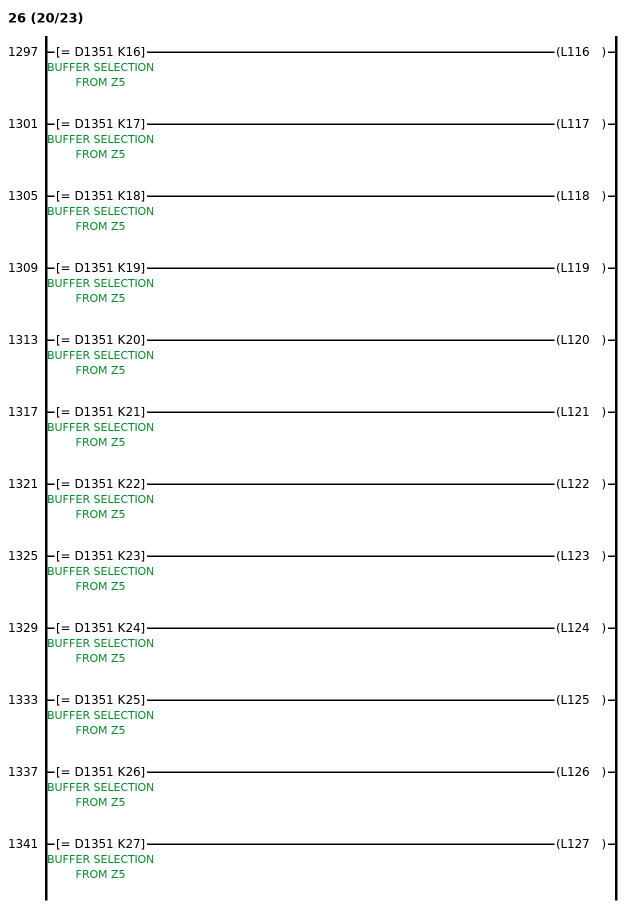
1297  LD=     D1351 K16  ; BUFFER SELECTION FROM Z5
      OUT     L116
1301  LD=     D1351 K17  ; BUFFER SELECTION FROM Z5
      OUT     L117
1305  LD=     D1351 K18  ; BUFFER SELECTION FROM Z5
      OUT     L118
1309  LD=     D1351 K19  ; BUFFER SELECTION FROM Z5
      OUT     L119
1313  LD=     D1351 K20  ; BUFFER SELECTION FROM Z5
      OUT     L120
1317  LD=     D1351 K21  ; BUFFER SELECTION FROM Z5
      OUT     L121
1321  LD=     D1351 K22  ; BUFFER SELECTION FROM Z5
      OUT     L122
1325  LD=     D1351 K23  ; BUFFER SELECTION FROM Z5
      OUT     L123
1329  LD=     D1351 K24  ; BUFFER SELECTION FROM Z5
      OUT     L124
1333  LD=     D1351 K25  ; BUFFER SELECTION FROM Z5
      OUT     L125
1337  LD=     D1351 K26  ; BUFFER SELECTION FROM Z5
      OUT     L126
1341  LD=     D1351 K27  ; BUFFER SELECTION FROM Z5
      OUT     L127
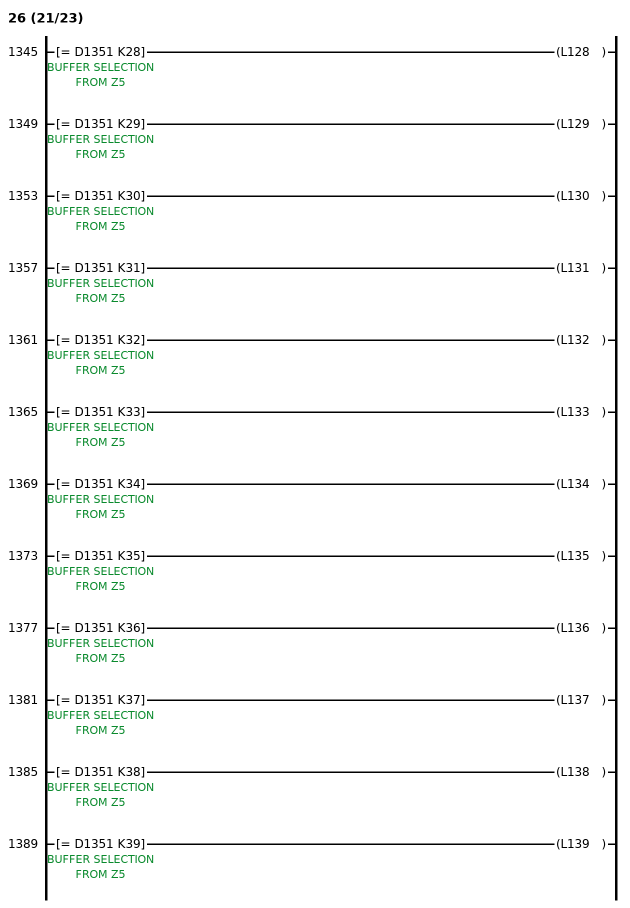
1345  LD=     D1351 K28  ; BUFFER SELECTION FROM Z5
      OUT     L128
1349  LD=     D1351 K29  ; BUFFER SELECTION FROM Z5
      OUT     L129
1353  LD=     D1351 K30  ; BUFFER SELECTION FROM Z5
      OUT     L130
1357  LD=     D1351 K31  ; BUFFER SELECTION FROM Z5
      OUT     L131
1361  LD=     D1351 K32  ; BUFFER SELECTION FROM Z5
      OUT     L132
1365  LD=     D1351 K33  ; BUFFER SELECTION FROM Z5
      OUT     L133
1369  LD=     D1351 K34  ; BUFFER SELECTION FROM Z5
      OUT     L134
1373  LD=     D1351 K35  ; BUFFER SELECTION FROM Z5
      OUT     L135
1377  LD=     D1351 K36  ; BUFFER SELECTION FROM Z5
      OUT     L136
1381  LD=     D1351 K37  ; BUFFER SELECTION FROM Z5
      OUT     L137
1385  LD=     D1351 K38  ; BUFFER SELECTION FROM Z5
      OUT     L138
1389  LD=     D1351 K39  ; BUFFER SELECTION FROM Z5
      OUT     L139
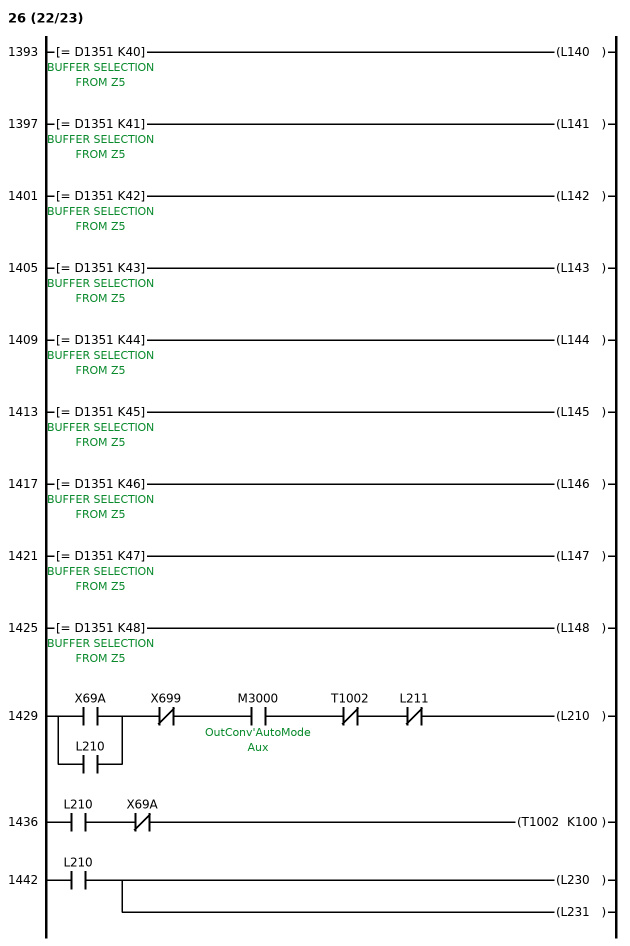
1393  LD=     D1351 K40  ; BUFFER SELECTION FROM Z5
      OUT     L140
1397  LD=     D1351 K41  ; BUFFER SELECTION FROM Z5
      OUT     L141
1401  LD=     D1351 K42  ; BUFFER SELECTION FROM Z5
      OUT     L142
1405  LD=     D1351 K43  ; BUFFER SELECTION FROM Z5
      OUT     L143
1409  LD=     D1351 K44  ; BUFFER SELECTION FROM Z5
      OUT     L144
1413  LD=     D1351 K45  ; BUFFER SELECTION FROM Z5
      OUT     L145
1417  LD=     D1351 K46  ; BUFFER SELECTION FROM Z5
      OUT     L146
1421  LD=     D1351 K47  ; BUFFER SELECTION FROM Z5
      OUT     L147
1425  LD=     D1351 K48  ; BUFFER SELECTION FROM Z5
      OUT     L148
1429  LD      X69A
      OR      L210
      ANI     X699
      AND     M3000  ; OutConv'AutoModeAux
      ANI     T1002
      ANI     L211
      OUT     L210
1436  LD      L210
      ANI     X69A
      OUT     T1002 K100
1442  LD      L210
      OUT     L230
      OUT     L231
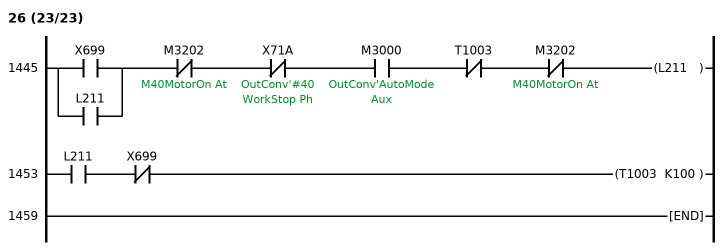
1445  LD      X699
      OR      L211
      ANI     M3202  ; M40MotorOn At
      ANI     X71A  ; OutConv'#40 WorkStop Ph
      AND     M3000  ; OutConv'AutoModeAux
      ANI     T1003
      ANI     M3202  ; M40MotorOn At
      OUT     L211
1453  LD      L211
      ANI     X699
      OUT     T1003 K100
1459  END
END_PROGRAM

PROGRAM 30  // Cycle Time
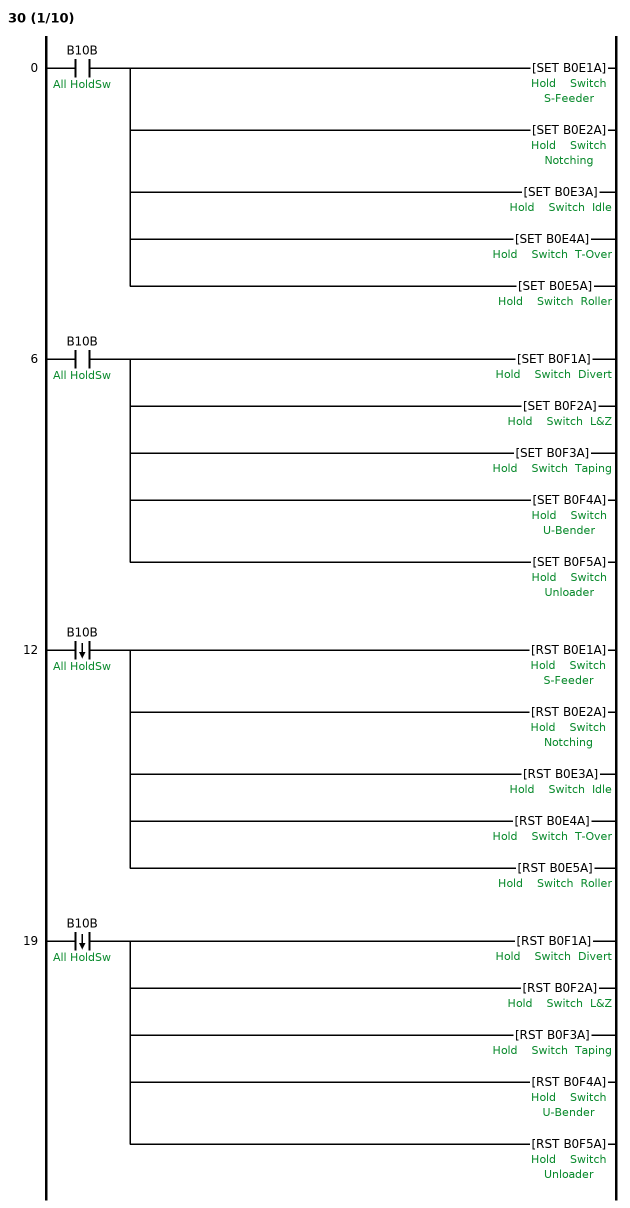
0     LD      B10B  ; All HoldSw
      SET     B0E1A  ; Hold    Switch  S-Feeder
      SET     B0E2A  ; Hold    Switch  Notching
      SET     B0E3A  ; Hold    Switch  Idle
      SET     B0E4A  ; Hold    Switch  T-Over
      SET     B0E5A  ; Hold    Switch  Roller
6     LD      B10B  ; All HoldSw
      SET     B0F1A  ; Hold    Switch  Divert
      SET     B0F2A  ; Hold    Switch  L&Z
      SET     B0F3A  ; Hold    Switch  Taping
      SET     B0F4A  ; Hold    Switch  U-Bender
      SET     B0F5A  ; Hold    Switch  Unloader
12    LDF     B10B  ; All HoldSw
      RST     B0E1A  ; Hold    Switch  S-Feeder
      RST     B0E2A  ; Hold    Switch  Notching
      RST     B0E3A  ; Hold    Switch  Idle
      RST     B0E4A  ; Hold    Switch  T-Over
      RST     B0E5A  ; Hold    Switch  Roller
19    LDF     B10B  ; All HoldSw
      RST     B0F1A  ; Hold    Switch  Divert
      RST     B0F2A  ; Hold    Switch  L&Z
      RST     B0F3A  ; Hold    Switch  Taping
      RST     B0F4A  ; Hold    Switch  U-Bender
      RST     B0F5A  ; Hold    Switch  Unloader
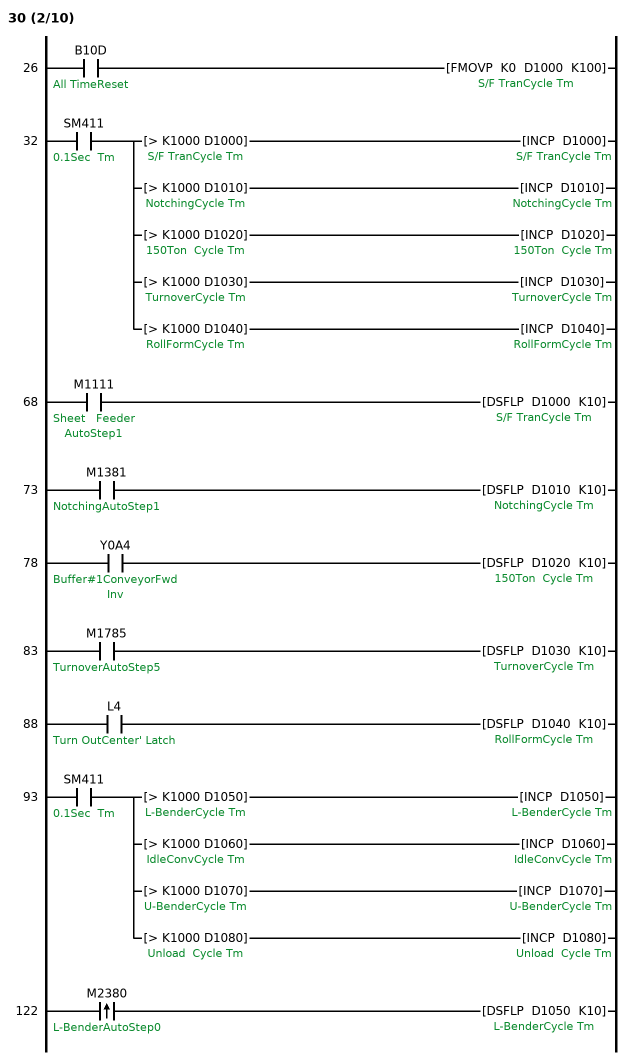
26    LD      B10D  ; All TimeReset
      FMOVP   K0 D1000 K100  ; S/F TranCycle Tm
32    LD      SM411  ; 0.1Sec  Tm
      MPS
      AND>    K1000 D1000  ; S/F TranCycle Tm
      INCP    D1000
      MRD
      AND>    K1000 D1010  ; NotchingCycle Tm
      INCP    D1010
      MRD
      AND>    K1000 D1020  ; 150Ton  Cycle Tm
      INCP    D1020
      MRD
      AND>    K1000 D1030  ; TurnoverCycle Tm
      INCP    D1030
      MPP
      AND>    K1000 D1040  ; RollFormCycle Tm
      INCP    D1040
68    LD      M1111  ; Sheet   Feeder  AutoStep1
      DSFLP   D1000 K10
73    LD      M1381  ; NotchingAutoStep1
      DSFLP   D1010 K10
78    LD      Y0A4  ; Buffer#1ConveyorFwd Inv
      DSFLP   D1020 K10
83    LD      M1785  ; TurnoverAutoStep5
      DSFLP   D1030 K10
88    LD      L4  ; Turn OutCenter' Latch
      DSFLP   D1040 K10
93    LD      SM411  ; 0.1Sec  Tm
      MPS
      AND>    K1000 D1050  ; L-BenderCycle Tm
      INCP    D1050
      MRD
      AND>    K1000 D1060  ; IdleConvCycle Tm
      INCP    D1060
      MRD
      AND>    K1000 D1070  ; U-BenderCycle Tm
      INCP    D1070
      MPP
      AND>    K1000 D1080  ; Unload  Cycle Tm
      INCP    D1080
122   LDP     M2380  ; L-BenderAutoStep0
      DSFLP   D1050 K10
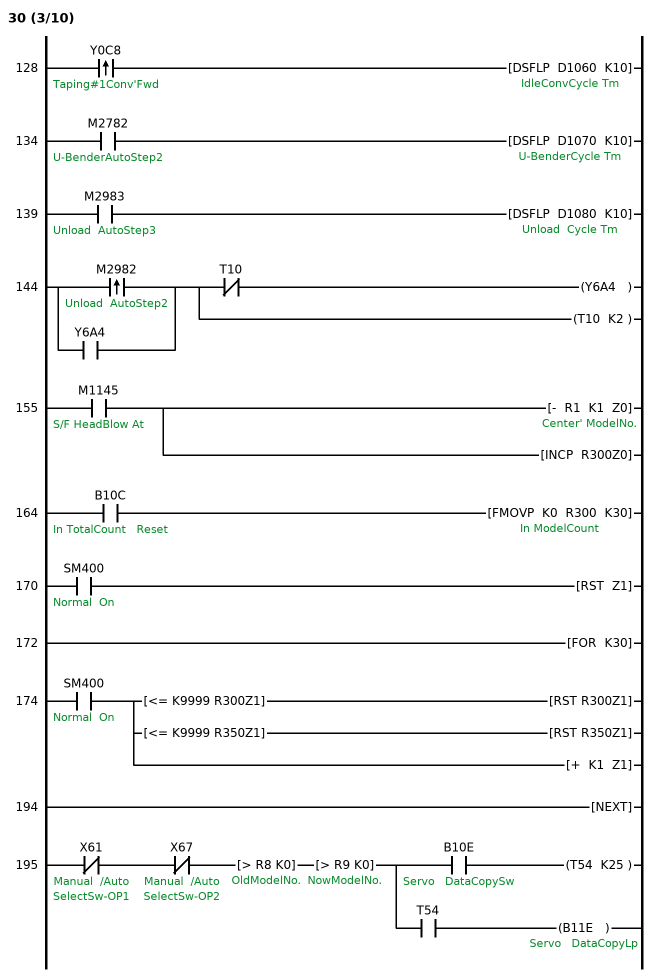
128   LDP     Y0C8  ; Taping#1Conv'Fwd
      DSFLP   D1060 K10
134   LD      M2782  ; U-BenderAutoStep2
      DSFLP   D1070 K10
139   LD      M2983  ; Unload  AutoStep3
      DSFLP   D1080 K10
144   LDP     M2982  ; Unload  AutoStep2
      OR      Y6A4
      MPS
      ANI     T10
      OUT     Y6A4
      MPP
      OUT     T10 K2
155   LD      M1145  ; S/F HeadBlow At
      -       R1 K1 Z0  ; Center' ModelNo.
      INCP    R300Z0
164   LD      B10C  ; In TotalCount   Reset
      FMOVP   K0 R300 K30  ; In ModelCount
170   LD      SM400  ; Normal  On
      RST     Z1
172   FOR     K30
174   LD      SM400  ; Normal  On
      MPS
      AND<=   K9999 R300Z1
      RST     R300Z1
      MRD
      AND<=   K9999 R350Z1
      RST     R350Z1
      MPP
      +       K1 Z1
194   NEXT
195   LDI     X61  ; Manual  /Auto   SelectSw-OP1
      ANI     X67  ; Manual  /Auto   SelectSw-OP2
      AND>    R8 K0  ; OldModelNo.
      AND>    R9 K0  ; NowModelNo.
      MPS
      AND     B10E  ; Servo   DataCopySw
      OUT     T54 K25
      MPP
      AND     T54
      OUT     B11E  ; Servo   DataCopyLp
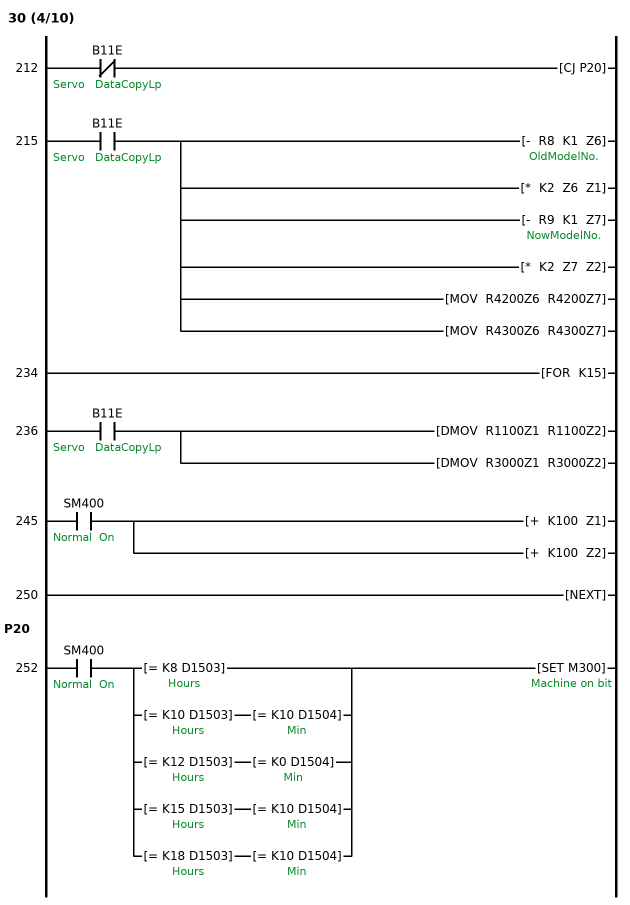
212   LDI     B11E  ; Servo   DataCopyLp
      CJ      P20
215   LD      B11E  ; Servo   DataCopyLp
      -       R8 K1 Z6
      *       K2 Z6 Z1
      -       R9 K1 Z7
      *       K2 Z7 Z2
      MOV     R4200Z6 R4200Z7
      MOV     R4300Z6 R4300Z7
234   FOR     K15
236   LD      B11E  ; Servo   DataCopyLp
      DMOV    R1100Z1 R1100Z2
      DMOV    R3000Z1 R3000Z2
245   LD      SM400  ; Normal  On
      +       K100 Z1
      +       K100 Z2
250   NEXT
      P20
252   LD      SM400  ; Normal  On
      LD=     K8 D1503  ; Hours
      LD=     K10 D1503  ; Hours
      AND=    K10 D1504  ; Min
      ORB
      LD=     K12 D1503  ; Hours
      AND=    K0 D1504  ; Min
      ORB
      LD=     K15 D1503  ; Hours
      AND=    K10 D1504  ; Min
      ORB
      LD=     K18 D1503  ; Hours
      AND=    K10 D1504  ; Min
      ORB
      ANB
      SET     M300  ; Machine on bit
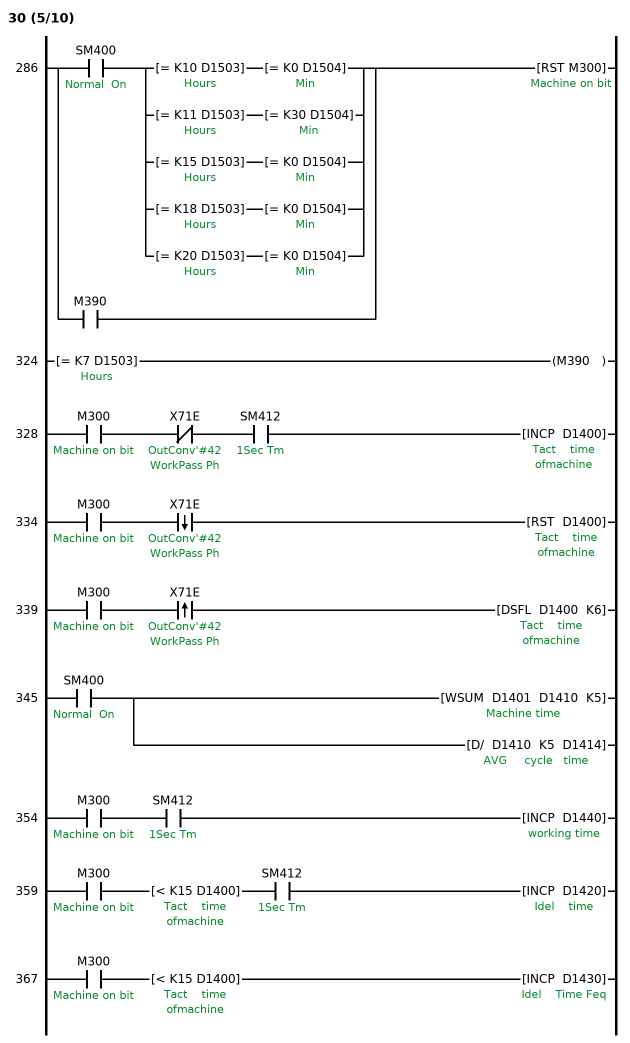
286   LD      SM400  ; Normal  On
      LD=     K10 D1503  ; Hours
      AND=    K0 D1504  ; Min
      LD=     K11 D1503  ; Hours
      AND=    K30 D1504  ; Min
      ORB
      LD=     K15 D1503  ; Hours
      AND=    K0 D1504  ; Min
      ORB
      LD=     K18 D1503  ; Hours
      AND=    K0 D1504  ; Min
      ORB
      LD=     K20 D1503  ; Hours
      AND=    K0 D1504  ; Min
      ORB
      ANB
      OR      M390
      RST     M300  ; Machine on bit
324   LD=     K7 D1503  ; Hours
      OUT     M390
328   LD      M300  ; Machine on bit
      ANI     X71E  ; OutConv'#42 WorkPass Ph
      AND     SM412  ; 1Sec Tm
      INCP    D1400  ; Tact    time  ofmachine
334   LD      M300  ; Machine on bit
      ANDF    X71E  ; OutConv'#42 WorkPass Ph
      RST     D1400  ; Tact    time  ofmachine
339   LD      M300  ; Machine on bit
      ANDP    X71E  ; OutConv'#42 WorkPass Ph
      DSFL    D1400 K6
345   LD      SM400  ; Normal  On
      WSUM    D1401 D1410 K5  ; Machine time
      D/      D1410 K5 D1414  ; AVG     cycle   time
354   LD      M300  ; Machine on bit
      AND     SM412  ; 1Sec Tm
      INCP    D1440  ; working time
359   LD      M300  ; Machine on bit
      AND<    K15 D1400  ; Tact    time  ofmachine
      AND     SM412  ; 1Sec Tm
      INCP    D1420  ; Idel    time
367   LD      M300  ; Machine on bit
      AND<    K15 D1400  ; Tact    time  ofmachine
      INCP    D1430  ; Idel    Time Feq
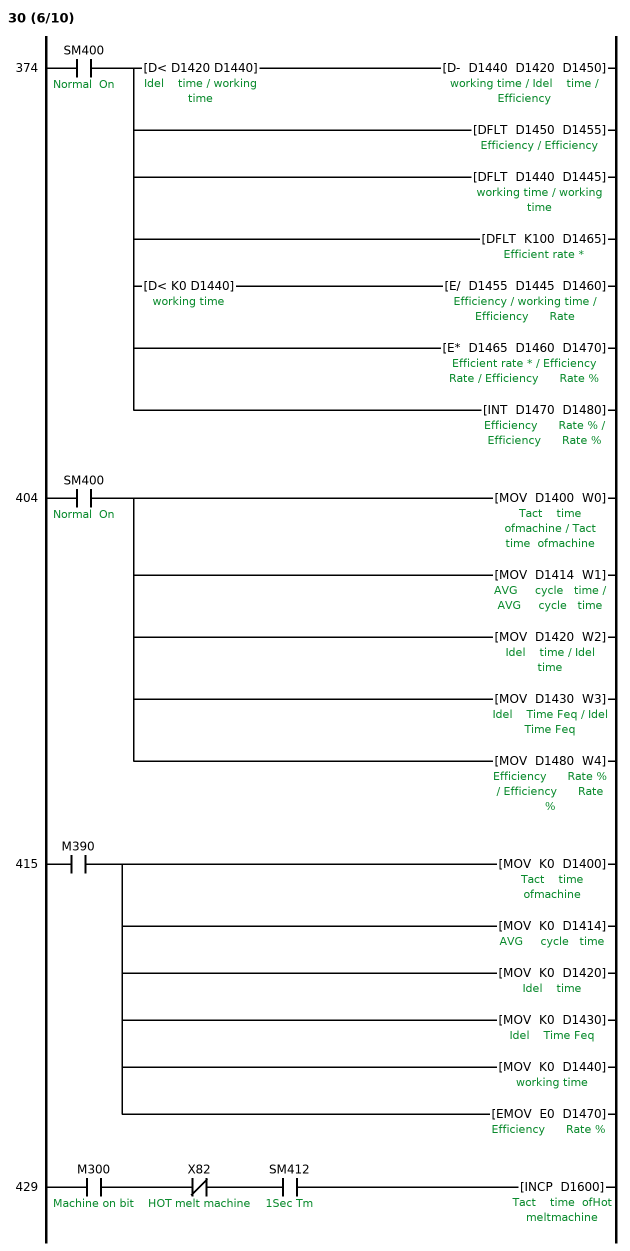
374   LD      SM400  ; Normal  On
      MPS
      ANDD<   D1420 D1440  ; Idel    time / working time
      D-      D1440 D1420 D1450  ; Efficiency
      MPP
      DFLT    D1450 D1455  ; Efficiency
      DFLT    D1440 D1445  ; working time
      DFLT    K100 D1465  ; Efficient rate *
      MPS
      ANDD<   K0 D1440  ; working time
      E/      D1455 D1445 D1460  ; Efficiency      Rate
      MPP
      E*      D1465 D1460 D1470  ; Efficiency      Rate %
      INT     D1470 D1480  ; Efficiency      Rate %
404   LD      SM400  ; Normal  On
      MOV     D1400 W0  ; Tact    time  ofmachine
      MOV     D1414 W1  ; AVG     cycle   time
      MOV     D1420 W2  ; Idel    time
      MOV     D1430 W3  ; Idel    Time Feq
      MOV     D1480 W4  ; Efficiency      Rate %
415   LD      M390
      MOV     K0 D1400
      MOV     K0 D1414
      MOV     K0 D1420
      MOV     K0 D1430
      MOV     K0 D1440
      EMOV    E0 D1470
429   LD      M300  ; Machine on bit
      ANI     X82  ; HOT melt machine
      AND     SM412  ; 1Sec Tm
      INCP    D1600  ; Tact    time  ofHot meltmachine
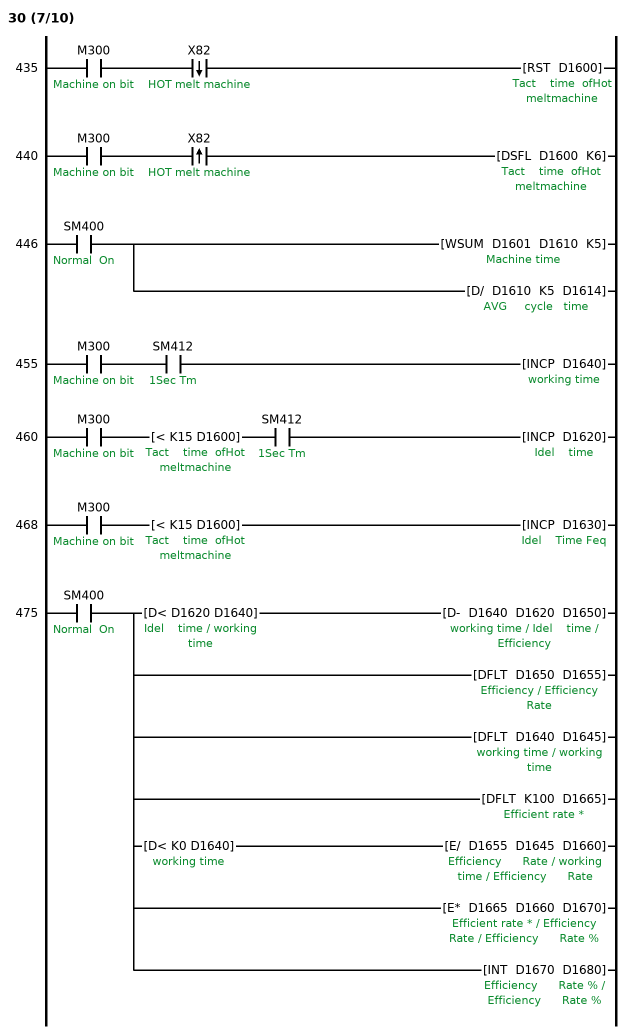
435   LD      M300  ; Machine on bit
      ANDF    X82  ; HOT melt machine
      RST     D1600  ; Tact    time  ofHot meltmachine
440   LD      M300  ; Machine on bit
      ANDP    X82  ; HOT melt machine
      DSFL    D1600 K6
446   LD      SM400  ; Normal  On
      WSUM    D1601 D1610 K5  ; Machine time
      D/      D1610 K5 D1614  ; AVG     cycle   time
455   LD      M300  ; Machine on bit
      AND     SM412  ; 1Sec Tm
      INCP    D1640  ; working time
460   LD      M300  ; Machine on bit
      AND<    K15 D1600  ; Tact    time  ofHot meltmachine
      AND     SM412  ; 1Sec Tm
      INCP    D1620  ; Idel    time
468   LD      M300  ; Machine on bit
      AND<    K15 D1600  ; Tact    time  ofHot meltmachine
      INCP    D1630  ; Idel    Time Feq
475   LD      SM400  ; Normal  On
      MPS
      ANDD<   D1620 D1640  ; Idel    time / working time
      D-      D1640 D1620 D1650  ; Efficiency
      MPP
      DFLT    D1650 D1655  ; Efficiency      Rate
      DFLT    D1640 D1645  ; working time
      DFLT    K100 D1665  ; Efficient rate *
      MPS
      ANDD<   K0 D1640  ; working time
      E/      D1655 D1645 D1660  ; Efficiency      Rate
      MPP
      E*      D1665 D1660 D1670  ; Efficiency      Rate %
      INT     D1670 D1680  ; Efficiency      Rate %
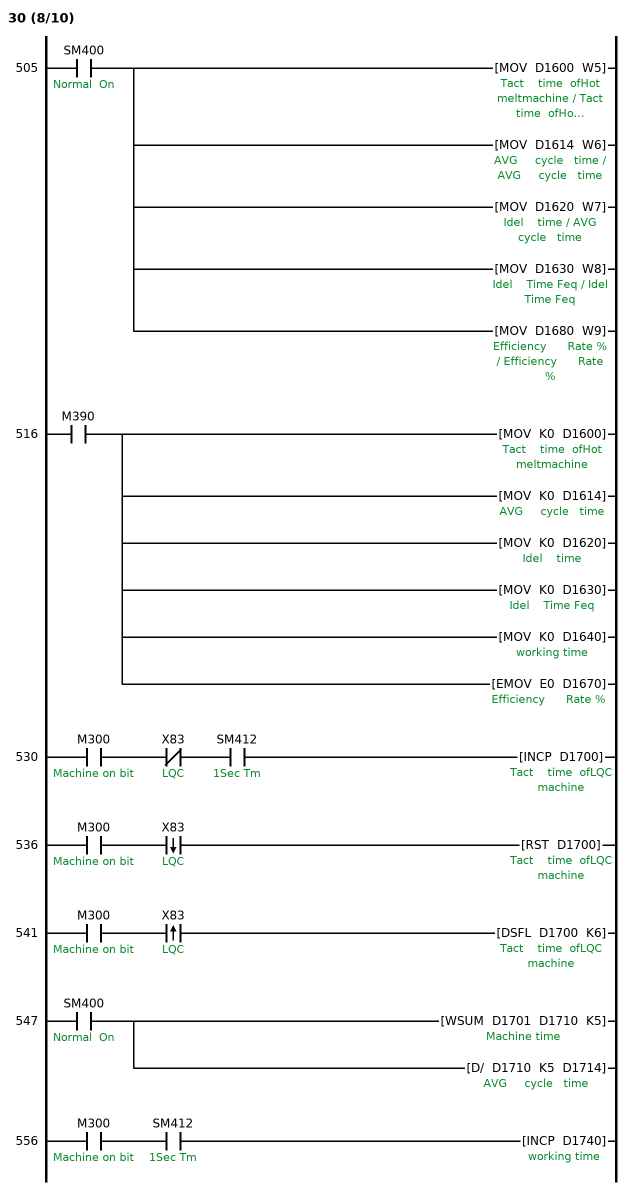
505   LD      SM400  ; Normal  On
      MOV     D1600 W5  ; Tact    time  ofHot meltmachine
      MOV     D1614 W6  ; AVG     cycle   time
      MOV     D1620 W7  ; AVG     cycle   time
      MOV     D1630 W8  ; Idel    Time Feq
      MOV     D1680 W9  ; Efficiency      Rate %
516   LD      M390
      MOV     K0 D1600
      MOV     K0 D1614
      MOV     K0 D1620
      MOV     K0 D1630
      MOV     K0 D1640
      EMOV    E0 D1670
530   LD      M300  ; Machine on bit
      ANI     X83  ; LQC
      AND     SM412  ; 1Sec Tm
      INCP    D1700  ; Tact    time  ofLQC     machine
536   LD      M300  ; Machine on bit
      ANDF    X83  ; LQC
      RST     D1700  ; Tact    time  ofLQC     machine
541   LD      M300  ; Machine on bit
      ANDP    X83  ; LQC
      DSFL    D1700 K6
547   LD      SM400  ; Normal  On
      WSUM    D1701 D1710 K5  ; Machine time
      D/      D1710 K5 D1714  ; AVG     cycle   time
556   LD      M300  ; Machine on bit
      AND     SM412  ; 1Sec Tm
      INCP    D1740  ; working time
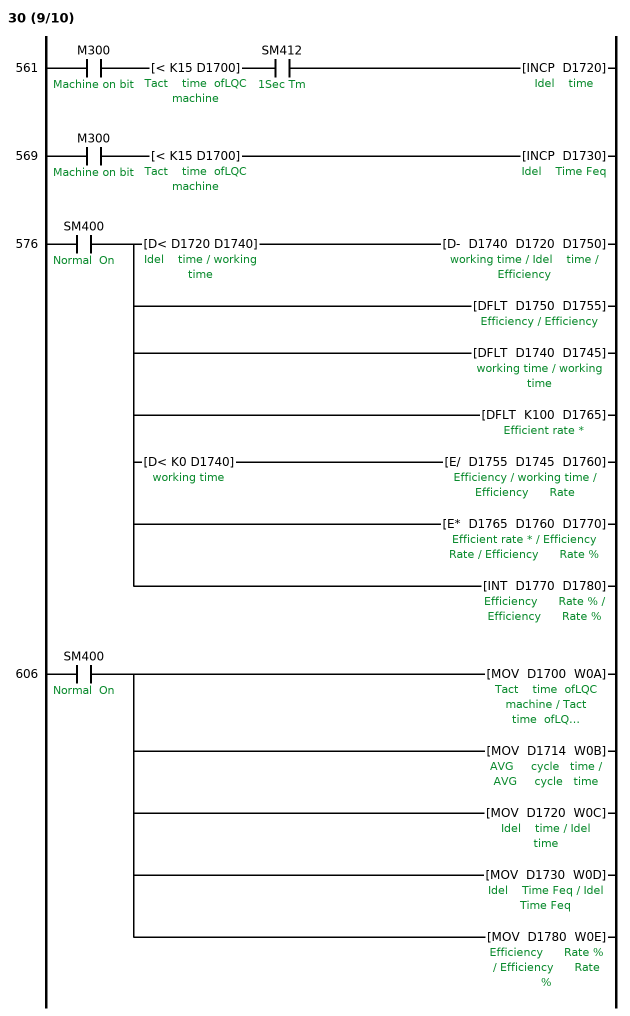
561   LD      M300  ; Machine on bit
      AND<    K15 D1700  ; Tact    time  ofLQC     machine
      AND     SM412  ; 1Sec Tm
      INCP    D1720  ; Idel    time
569   LD      M300  ; Machine on bit
      AND<    K15 D1700  ; Tact    time  ofLQC     machine
      INCP    D1730  ; Idel    Time Feq
576   LD      SM400  ; Normal  On
      MPS
      ANDD<   D1720 D1740  ; Idel    time / working time
      D-      D1740 D1720 D1750  ; Efficiency
      MPP
      DFLT    D1750 D1755  ; Efficiency
      DFLT    D1740 D1745  ; working time
      DFLT    K100 D1765  ; Efficient rate *
      MPS
      ANDD<   K0 D1740  ; working time
      E/      D1755 D1745 D1760  ; Efficiency      Rate
      MPP
      E*      D1765 D1760 D1770  ; Efficiency      Rate %
      INT     D1770 D1780  ; Efficiency      Rate %
606   LD      SM400  ; Normal  On
      MOV     D1700 W0A  ; Tact    time  ofLQC     machine
      MOV     D1714 W0B  ; AVG     cycle   time
      MOV     D1720 W0C  ; Idel    time
      MOV     D1730 W0D  ; Idel    Time Feq
      MOV     D1780 W0E  ; Efficiency      Rate %
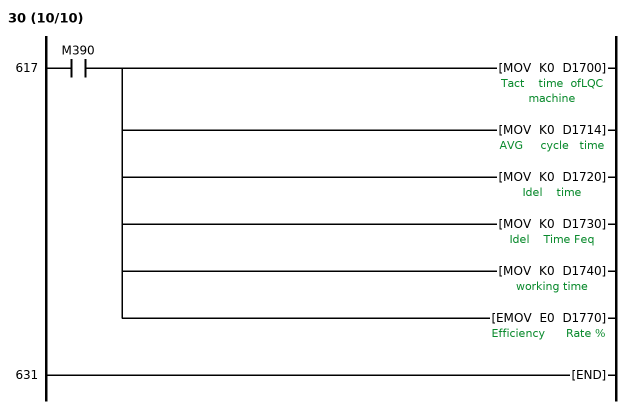
617   LD      M390
      MOV     K0 D1700
      MOV     K0 D1714
      MOV     K0 D1720
      MOV     K0 D1730
      MOV     K0 D1740
      EMOV    E0 D1770
631   END
END_PROGRAM

PROGRAM MAIN  // MAIN
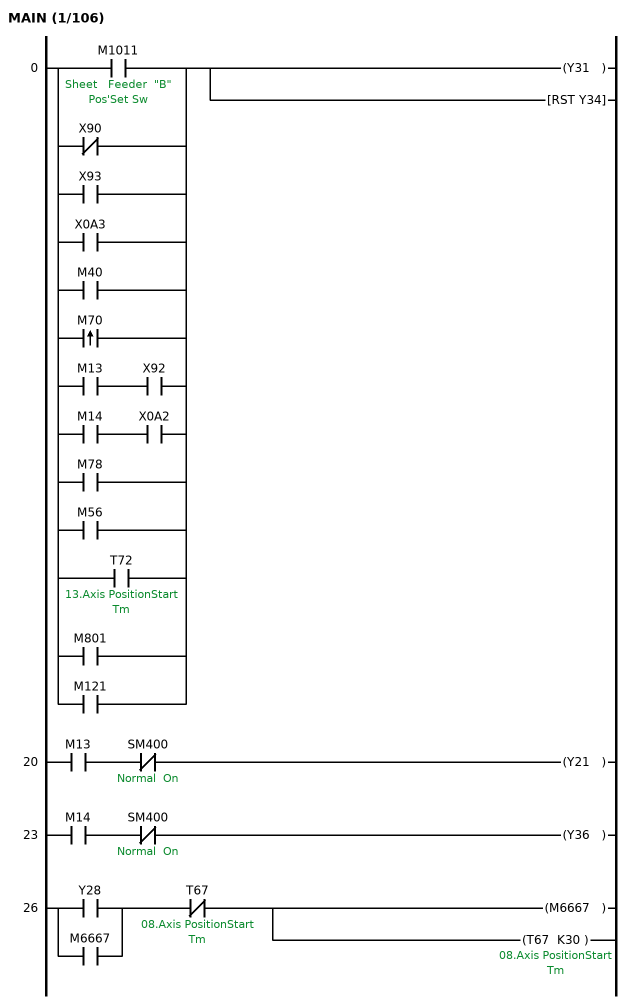
0     LD      M1011  ; Sheet   Feeder  "B" Pos'Set Sw
      ORI     X90
      OR      X93
      OR      X0A3
      OR      M40
      ORP     M70
      LD      M13
      AND     X92
      ORB
      LD      M14
      AND     X0A2
      ORB
      OR      M78
      OR      M56
      OR      T72  ; 13.Axis PositionStart Tm
      OR      M801
      OR      M121
      OUT     Y31
      RST     Y34
20    LD      M13
      ANI     SM400  ; Normal  On
      OUT     Y21
23    LD      M14
      ANI     SM400  ; Normal  On
      OUT     Y36
26    LD      Y28
      OR      M6667
      ANI     T67  ; 08.Axis PositionStart Tm
      OUT     M6667
      OUT     T67 K30  ; 08.Axis PositionStart Tm
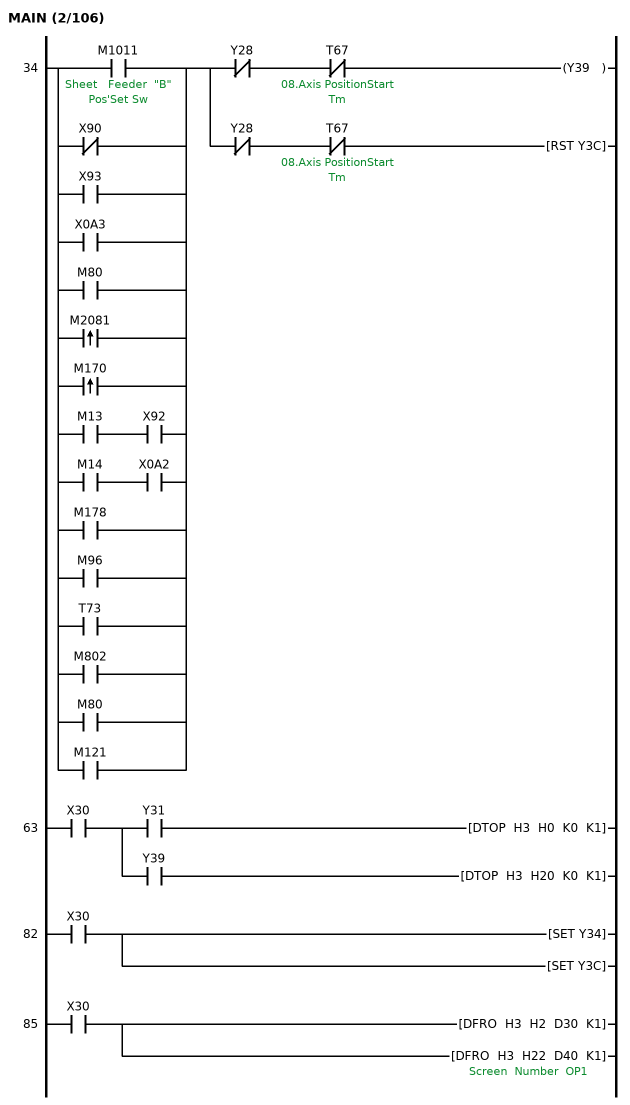
34    LD      M1011  ; Sheet   Feeder  "B" Pos'Set Sw
      ORI     X90
      OR      X93
      OR      X0A3
      OR      M80
      ORP     M2081
      ORP     M170
      LD      M13
      AND     X92
      ORB
      LD      M14
      AND     X0A2
      ORB
      OR      M178
      OR      M96
      OR      T73
      OR      M802
      OR      M80
      OR      M121
      MPS
      ANI     Y28
      ANI     T67  ; 08.Axis PositionStart Tm
      OUT     Y39
      MPP
      ANI     Y28
      ANI     T67  ; 08.Axis PositionStart Tm
      RST     Y3C
63    LD      X30
      MPS
      AND     Y31
      DTOP    H3 H0 K0 K1
      MPP
      AND     Y39
      DTOP    H3 H20 K0 K1
82    LD      X30
      SET     Y34
      SET     Y3C
85    LD      X30
      DFRO    H3 H2 D30 K1
      DFRO    H3 H22 D40 K1  ; Screen  Number  OP1
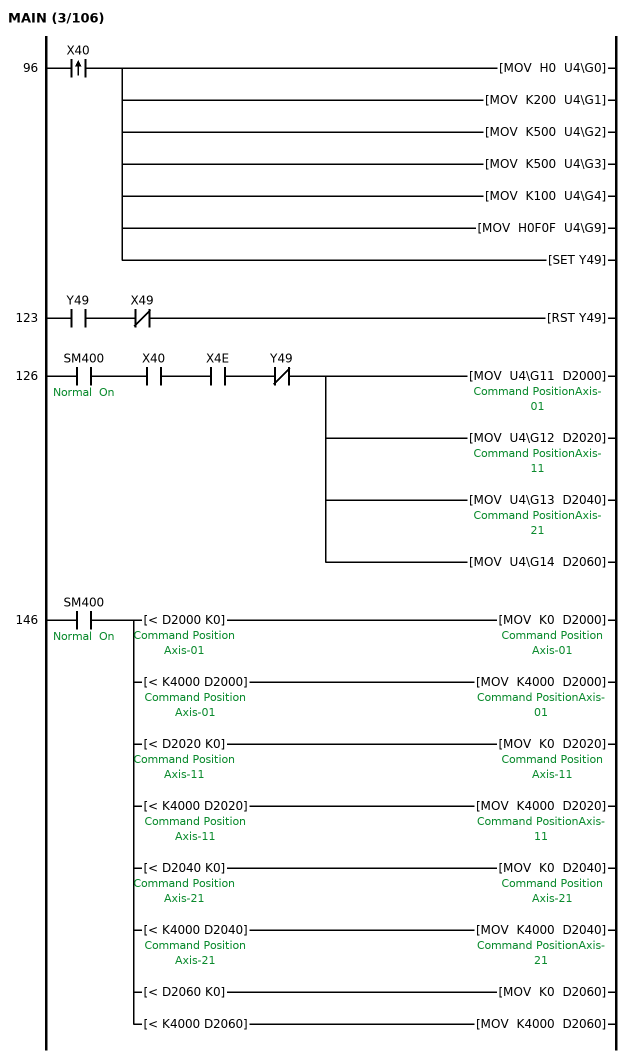
96    LDP     X40
      MOV     H0 U4\G0
      MOV     K200 U4\G1
      MOV     K500 U4\G2
      MOV     K500 U4\G3
      MOV     K100 U4\G4
      MOV     H0F0F U4\G9
      SET     Y49
123   LD      Y49
      ANI     X49
      RST     Y49
126   LD      SM400  ; Normal  On
      AND     X40
      AND     X4E
      ANI     Y49
      MOV     U4\G11 D2000  ; Command PositionAxis-01
      MOV     U4\G12 D2020  ; Command PositionAxis-11
      MOV     U4\G13 D2040  ; Command PositionAxis-21
      MOV     U4\G14 D2060
146   LD      SM400  ; Normal  On
      MPS
      AND<    D2000 K0  ; Command PositionAxis-01
      MOV     K0 D2000
      MRD
      AND<    K4000 D2000  ; Command PositionAxis-01
      MOV     K4000 D2000
      MRD
      AND<    D2020 K0  ; Command PositionAxis-11
      MOV     K0 D2020
      MRD
      AND<    K4000 D2020  ; Command PositionAxis-11
      MOV     K4000 D2020
      MRD
      AND<    D2040 K0  ; Command PositionAxis-21
      MOV     K0 D2040
      MRD
      AND<    K4000 D2040  ; Command PositionAxis-21
      MOV     K4000 D2040
      MRD
      AND<    D2060 K0
      MOV     K0 D2060
      MPP
      AND<    K4000 D2060
      MOV     K4000 D2060
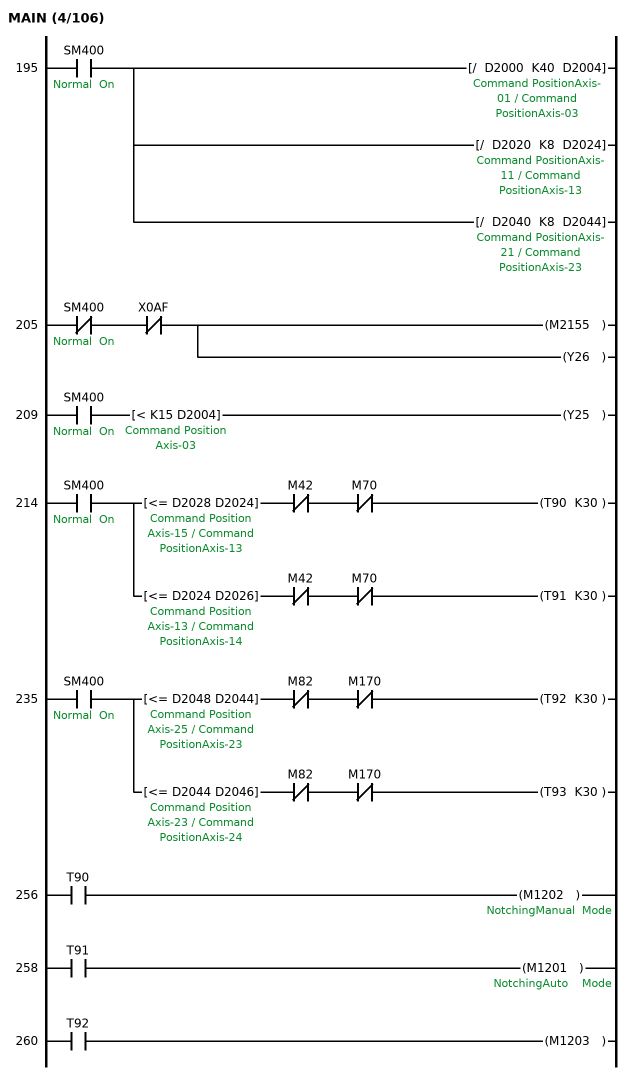
195   LD      SM400  ; Normal  On
      /       D2000 K40 D2004  ; Command PositionAxis-03
      /       D2020 K8 D2024  ; Command PositionAxis-13
      /       D2040 K8 D2044  ; Command PositionAxis-23
205   LDI     SM400  ; Normal  On
      ANI     X0AF
      OUT     M2155
      OUT     Y26
209   LD      SM400  ; Normal  On
      AND<    K15 D2004  ; Command PositionAxis-03
      OUT     Y25
214   LD      SM400  ; Normal  On
      MPS
      AND<=   D2028 D2024  ; Command PositionAxis-15 / Command PositionAxis-13
      ANI     M42
      ANI     M70
      OUT     T90 K30
      MPP
      AND<=   D2024 D2026  ; Command PositionAxis-13 / Command PositionAxis-14
      ANI     M42
      ANI     M70
      OUT     T91 K30
235   LD      SM400  ; Normal  On
      MPS
      AND<=   D2048 D2044  ; Command PositionAxis-25 / Command PositionAxis-23
      ANI     M82
      ANI     M170
      OUT     T92 K30
      MPP
      AND<=   D2044 D2046  ; Command PositionAxis-23 / Command PositionAxis-24
      ANI     M82
      ANI     M170
      OUT     T93 K30
256   LD      T90
      OUT     M1202  ; NotchingManual  Mode
258   LD      T91
      OUT     M1201  ; NotchingAuto    Mode
260   LD      T92
      OUT     M1203
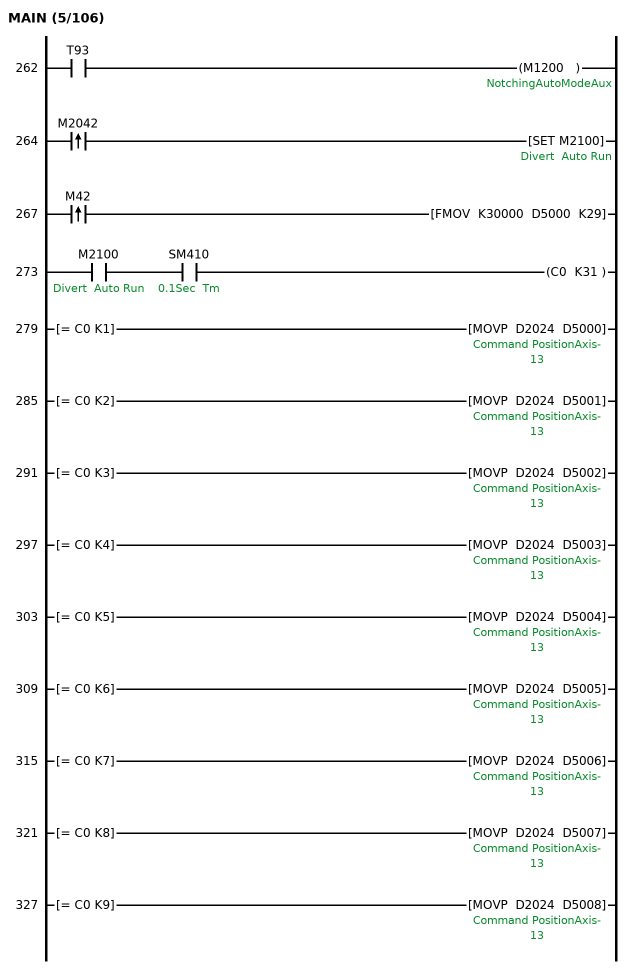
262   LD      T93
      OUT     M1200  ; NotchingAutoModeAux
264   LDP     M2042
      SET     M2100  ; Divert  Auto Run
267   LDP     M42
      FMOV    K30000 D5000 K29
273   LD      M2100  ; Divert  Auto Run
      AND     SM410  ; 0.1Sec  Tm
      OUT     C0 K31
279   LD=     C0 K1
      MOVP    D2024 D5000
285   LD=     C0 K2
      MOVP    D2024 D5001
291   LD=     C0 K3
      MOVP    D2024 D5002
297   LD=     C0 K4
      MOVP    D2024 D5003
303   LD=     C0 K5
      MOVP    D2024 D5004
309   LD=     C0 K6
      MOVP    D2024 D5005
315   LD=     C0 K7
      MOVP    D2024 D5006
321   LD=     C0 K8
      MOVP    D2024 D5007
327   LD=     C0 K9
      MOVP    D2024 D5008
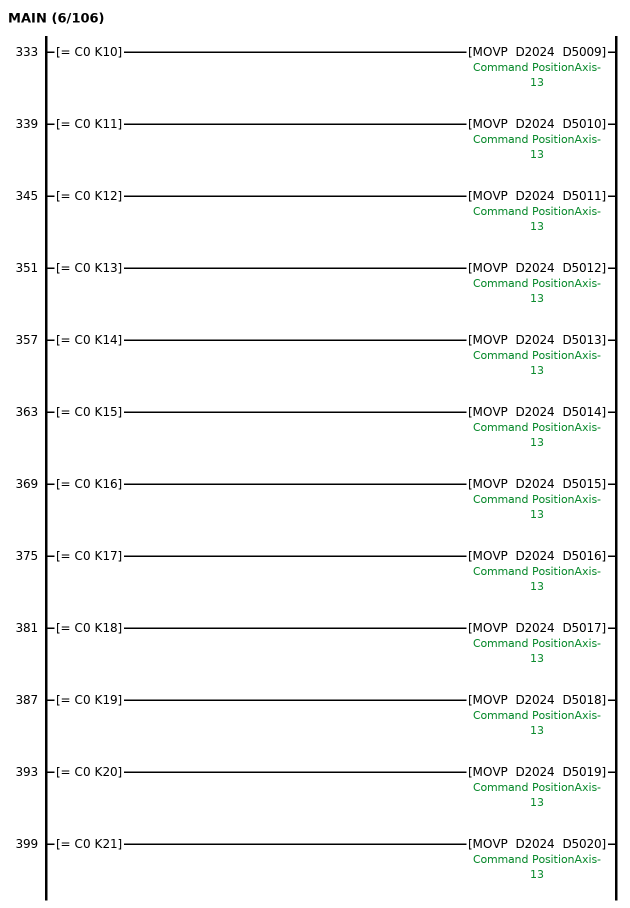
333   LD=     C0 K10
      MOVP    D2024 D5009
339   LD=     C0 K11
      MOVP    D2024 D5010
345   LD=     C0 K12
      MOVP    D2024 D5011
351   LD=     C0 K13
      MOVP    D2024 D5012
357   LD=     C0 K14
      MOVP    D2024 D5013
363   LD=     C0 K15
      MOVP    D2024 D5014
369   LD=     C0 K16
      MOVP    D2024 D5015
375   LD=     C0 K17
      MOVP    D2024 D5016
381   LD=     C0 K18
      MOVP    D2024 D5017
387   LD=     C0 K19
      MOVP    D2024 D5018
393   LD=     C0 K20
      MOVP    D2024 D5019
399   LD=     C0 K21
      MOVP    D2024 D5020
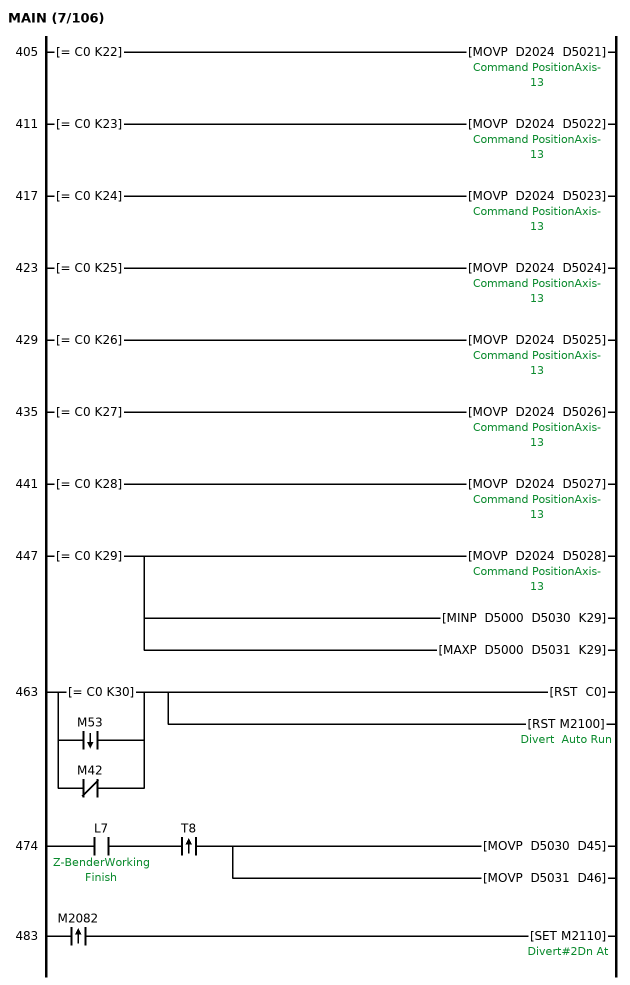
405   LD=     C0 K22
      MOVP    D2024 D5021
411   LD=     C0 K23
      MOVP    D2024 D5022
417   LD=     C0 K24
      MOVP    D2024 D5023
423   LD=     C0 K25
      MOVP    D2024 D5024
429   LD=     C0 K26
      MOVP    D2024 D5025
435   LD=     C0 K27
      MOVP    D2024 D5026
441   LD=     C0 K28
      MOVP    D2024 D5027
447   LD=     C0 K29
      MOVP    D2024 D5028
      MINP    D5000 D5030 K29
      MAXP    D5000 D5031 K29
463   LD=     C0 K30
      ORF     M53
      ORI     M42
      RST     C0
      RST     M2100  ; Divert  Auto Run
474   LD      L7  ; Z-BenderWorking Finish
      ANDP    T8
      MOVP    D5030 D45
      MOVP    D5031 D46
483   LDP     M2082
      SET     M2110  ; Divert#2Dn At
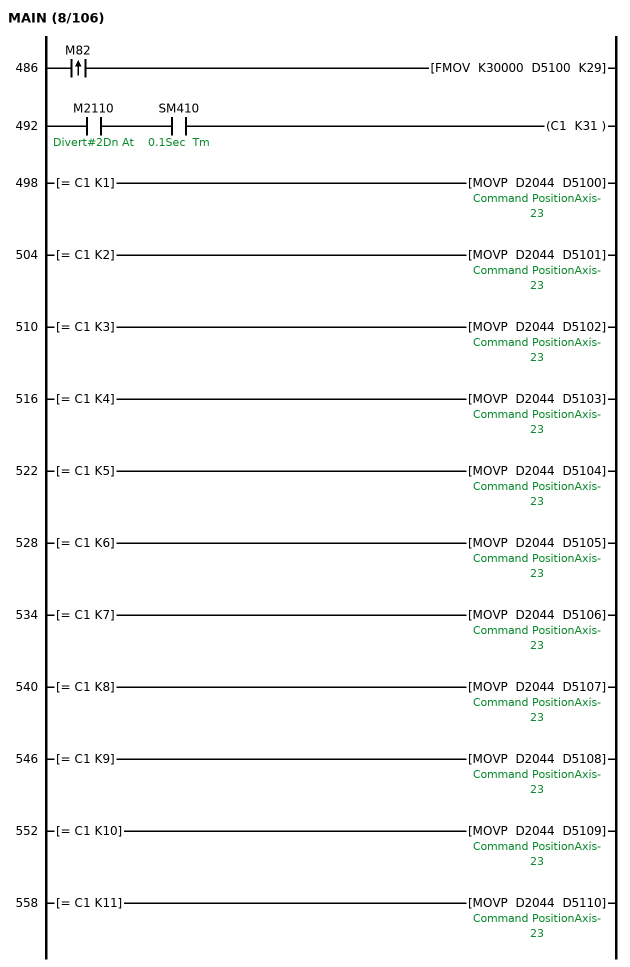
486   LDP     M82
      FMOV    K30000 D5100 K29
492   LD      M2110  ; Divert#2Dn At
      AND     SM410  ; 0.1Sec  Tm
      OUT     C1 K31
498   LD=     C1 K1
      MOVP    D2044 D5100
504   LD=     C1 K2
      MOVP    D2044 D5101
510   LD=     C1 K3
      MOVP    D2044 D5102
516   LD=     C1 K4
      MOVP    D2044 D5103
522   LD=     C1 K5
      MOVP    D2044 D5104
528   LD=     C1 K6
      MOVP    D2044 D5105
534   LD=     C1 K7
      MOVP    D2044 D5106
540   LD=     C1 K8
      MOVP    D2044 D5107
546   LD=     C1 K9
      MOVP    D2044 D5108
552   LD=     C1 K10
      MOVP    D2044 D5109
558   LD=     C1 K11
      MOVP    D2044 D5110
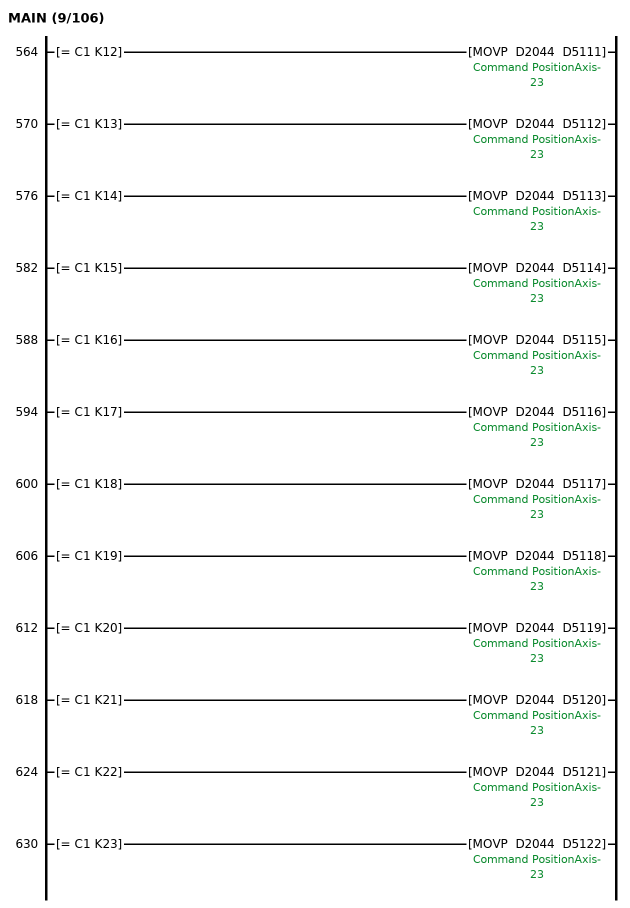
564   LD=     C1 K12
      MOVP    D2044 D5111
570   LD=     C1 K13
      MOVP    D2044 D5112
576   LD=     C1 K14
      MOVP    D2044 D5113
582   LD=     C1 K15
      MOVP    D2044 D5114
588   LD=     C1 K16
      MOVP    D2044 D5115
594   LD=     C1 K17
      MOVP    D2044 D5116
600   LD=     C1 K18
      MOVP    D2044 D5117
606   LD=     C1 K19
      MOVP    D2044 D5118
612   LD=     C1 K20
      MOVP    D2044 D5119
618   LD=     C1 K21
      MOVP    D2044 D5120
624   LD=     C1 K22
      MOVP    D2044 D5121
630   LD=     C1 K23
      MOVP    D2044 D5122
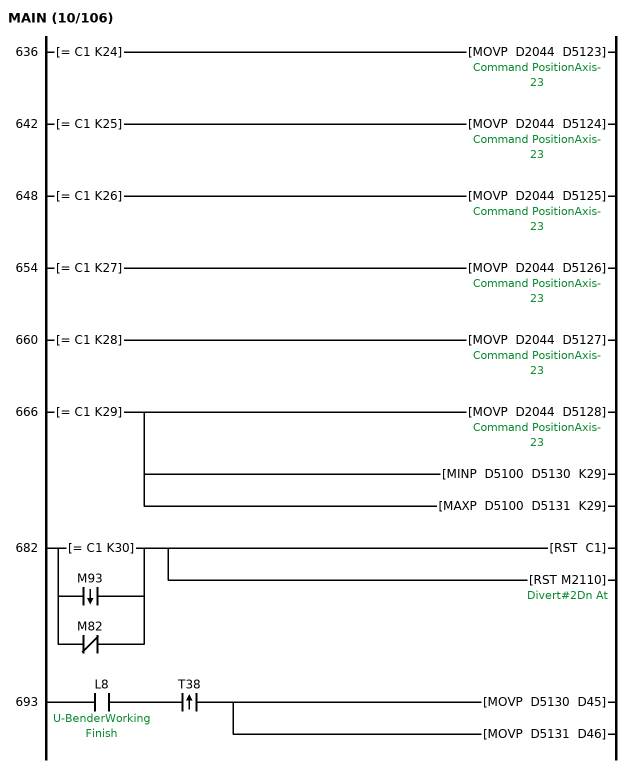
636   LD=     C1 K24
      MOVP    D2044 D5123
642   LD=     C1 K25
      MOVP    D2044 D5124
648   LD=     C1 K26
      MOVP    D2044 D5125
654   LD=     C1 K27
      MOVP    D2044 D5126
660   LD=     C1 K28
      MOVP    D2044 D5127
666   LD=     C1 K29
      MOVP    D2044 D5128
      MINP    D5100 D5130 K29
      MAXP    D5100 D5131 K29
682   LD=     C1 K30
      ORF     M93
      ORI     M82
      RST     C1
      RST     M2110  ; Divert#2Dn At
693   LD      L8  ; U-BenderWorking Finish
      ANDP    T38
      MOVP    D5130 D45
      MOVP    D5131 D46
